FUNCTION TryConvert_UDINT_TO_REAL : BOOL
VAR_INPUT
	in : UDINT;
	out : REFERENCE TO REAL;
END_VAR

out := UDINT_TO_REAL(in);
TryConvert_UDINT_TO_REAL := TRUE;

END_FUNCTION

(* stored: Version 1.1.0.1, ProductVersion 3.1.4024.12
   POU TryConvert_UDINT_TO_REAL: Id {1c26be60-a749-49ad-91d2-b97da079781f}, SpecialFunc None *)
